// SIMATIC S7-200 SMART project (STEP 7-Micro/WIN SMART), CPU ST40

SYMBOL_TABLE Table 1
Fill_Button      V0.0
Discharge_Button V0.1
Fill_Valve       Q0.0
Filling          Q0.1
Discharge_Valve  Q0.2
Discharging      Q0.3
Timer            QW4
Potentiometer    VW100
Emergency_Button V0.2
Scaled           VW108
END_SYMBOL_TABLE

SYMBOL_TABLE System Symbols
Always_On        SM0.0    // Always ON
END_SYMBOL_TABLE

ORGANIZATION_BLOCK MAIN:OB1
TITLE=Program Comments
BEGIN
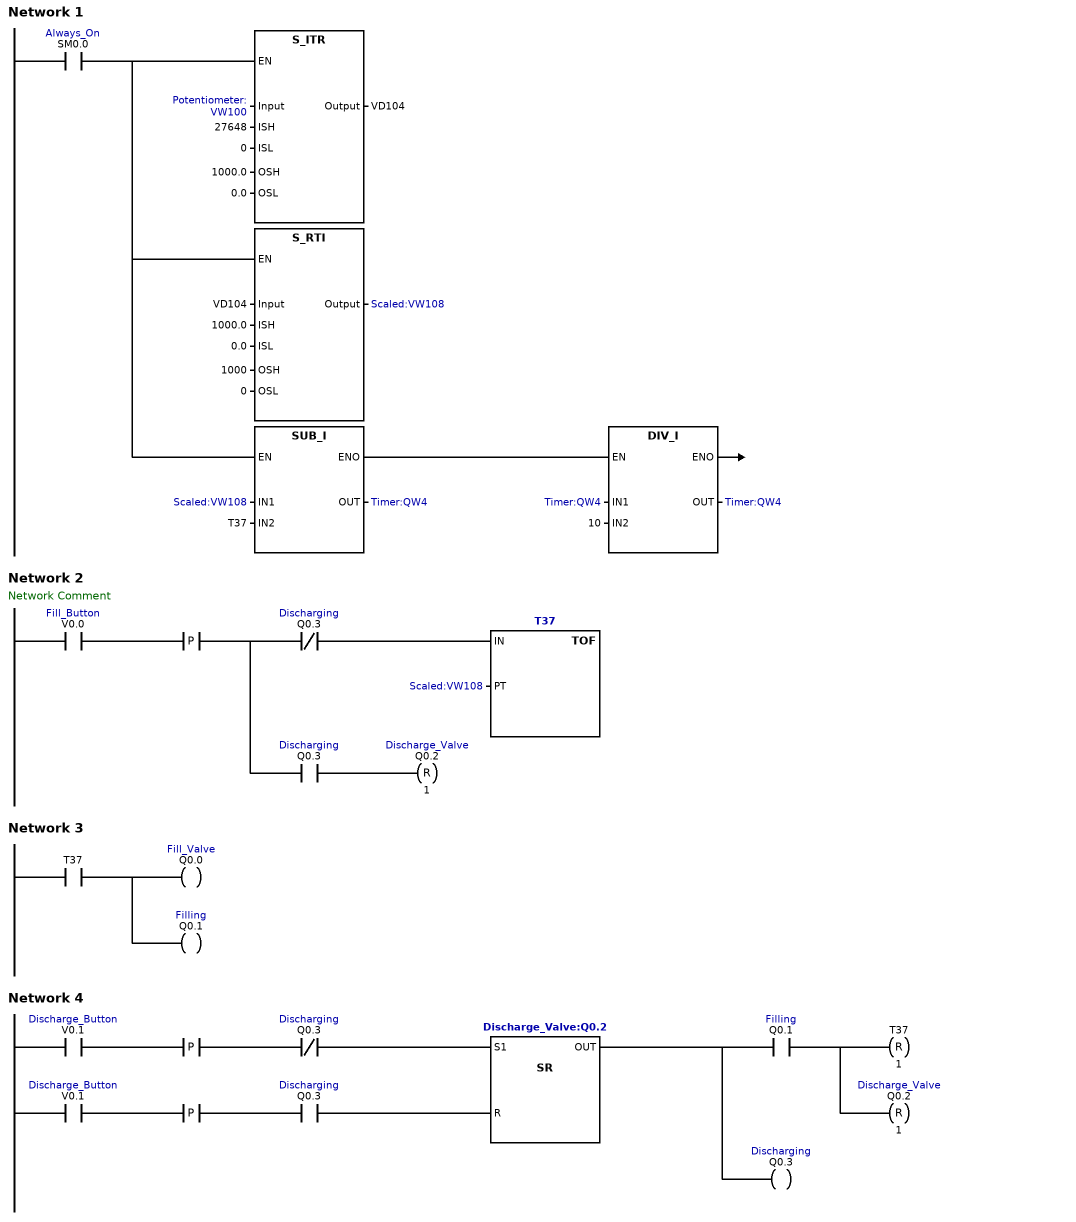
Network 1
LD     Always_On:SM0.0
CALL   S_ITR:SBR1, Potentiometer:VW100, 27648, 0, 1000.0, 0.0, VD104
CALL   S_RTI:SBR2, VD104, 1000.0, 0.0, 1000, 0, Scaled:VW108
MOVW   Scaled:VW108, Timer:QW4
AENO
-I     T37, Timer:QW4
AENO
/I     10, Timer:QW4
Network 2
// Network Comment
LD     Fill_Button:V0.0
EU
LPS
AN     Discharging:Q0.3
TOF    T37, Scaled:VW108
LPP
A      Discharging:Q0.3
R      Discharge_Valve:Q0.2, 1
Network 3
LD     T37
=      Fill_Valve:Q0.0
=      Filling:Q0.1
Network 4
LD     Discharge_Button:V0.1
EU
AN     Discharging:Q0.3
LD     Discharge_Button:V0.1
EU
A      Discharging:Q0.3
NOT
A      Discharge_Valve:Q0.2
OLD
=      Discharge_Valve:Q0.2
LPS
A      Filling:Q0.1
R      T37, 1
R      Discharge_Valve:Q0.2, 1
LPP
=      Discharging:Q0.3
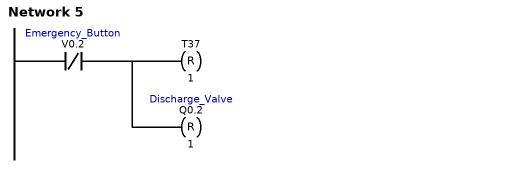
Network 5
LDN    Emergency_Button:V0.2
R      T37, 1
R      Discharge_Valve:Q0.2, 1
END_ORGANIZATION_BLOCK

// SBR1: protected block, not included

// SBR2: protected block, not included

// (further data pages could not be read)
